INTERFACE I_Mc2MotionTaskCollection EXTENDS I_MotionTaskCollection

METHOD AddTask
VAR_INPUT
	Task : I_Mc2MotionTask;
END_VAR
END_METHOD

METHOD RemoveTaskByInstance
VAR_INPUT
	Task : I_Mc2MotionTask;
END_VAR
END_METHOD

END_INTERFACE

(* stored: Version 1.1.0.1, ProductVersion 3.1.4026.20
   Itf I_Mc2MotionTaskCollection: Id {5cef30fa-20ec-45a3-9abb-6d3952f0de91}
   Method AddTask: Id {2950274e-7e92-4b87-8014-c41a77a99a45}
   Method RemoveTaskByInstance: Id {7678a5bd-5735-492c-a995-a537ca3df1bd} *)
